(* PLC project mtcs_services, Institute of Astronomy OntoManager 0.0.1 *)
(* stored: creationDateTime 2017-02-05T17:05:48.277559, modificationDateTime 2017-02-05T17:05:48.277559 *)

TYPE ServicesTimingTimeSource : (LOCAL_CLOCK := 0, PTP_IEEE_1588 := 1);
END_TYPE

TYPE ServicesMeteoId : (WIND_SPEED_MINIMUM := 0, WIND_SPEED_AVERAGE := 1, WIND_SPEED_MAXIMUM := 2, WIND_DIRECTION_MINIMUM := 3, WIND_DIRECTION_AVERAGE := 4, WIND_DIRECTION_MAXIMUM := 5, AIR_PRESSURE := 6, AIR_TEMPERATURE := 7, INTERNAL_TEMPERATURE := 8, RELATIVE_HUMIDITY := 9, RAIN_ACCUMULATION := 10, RAIN_DURATION := 11, RAIN_INTENSITY := 12, RAIN_PEAK_INTENSITY := 13, HAIL_ACCUMULATION := 14, HAIL_DURATION := 15, HAIL_PEAK_INTENSITY := 16, HAIL_INTENSITY := 17, HEATING_TEMPERATURE := 18, HEATING_VOLTAGE := 19, SUPPLY_VOLTAGE := 20, REFERENCE_VOLTAGE := 21);
END_TYPE

TYPE ServicesParts : STRUCT
  timing : ServicesTiming;  (* Timing service *)
  meteo : ServicesMeteo;  (* Meteo service *)
  io : ServicesIO;  (* I/O modules *)
  configManager : ConfigManager;  (* The config manager (to load/save/activate configuration data) *)
END_STRUCT;
END_TYPE

TYPE ServicesTimingParts : STRUCT
  serialInfo : ServicesTimingSerialInfo;  (* Info acquired by serial link *)
END_STRUCT;
END_TYPE

TYPE ServicesIOParts : STRUCT
  coupler : EtherCatDevice;  (* Coupler *)
  slot1 : EtherCatDevice;  (* Slot 1 *)
  slot2 : EtherCatDevice;  (* Slot 2 *)
  slot3 : EtherCatDevice;  (* Slot 2 *)
END_STRUCT;
END_TYPE

TYPE ServicesProcesses : STRUCT
  initialize : Process;  (* Start initializing *)
  lock : Process;  (* Lock the system *)
  unlock : Process;  (* Unlock the system *)
  changeOperatingState : ChangeOperatingStateProcess;  (* Change the operating state (e.g. AUTO, MANUAL, ...) *)
END_STRUCT;
END_TYPE

TYPE ServicesTimingProcesses : STRUCT

END_STRUCT;
END_TYPE

TYPE ServicesMeteoProcesses : STRUCT

END_STRUCT;
END_TYPE

TYPE ServicesStatuses : STRUCT
  initializationStatus : InitializationStatus;
  healthStatus : HealthStatus;
  busyStatus : BusyStatus;
  operatingStatus : OperatingStatus;
END_STRUCT;
END_TYPE

TYPE ServicesTimingStatuses : STRUCT
  healthStatus : HealthStatus;
END_STRUCT;
END_TYPE

TYPE ServicesTimingSerialInfoStatuses : STRUCT
  portHealthStatus : HealthStatus;
  transmissionHealthStatus : HealthStatus;
  checksumHealthStatus : HealthStatus;
  healthStatus : HealthStatus;
END_STRUCT;
END_TYPE

TYPE ServicesMeteoMeasurementStatuses : STRUCT
  enabledStatus : EnabledStatus;  (* Is the temperature being measured? *)
  healthStatus : HealthStatus;  (* Is the data valid and within range? *)
  alarmStatus : HiHiLoLoAlarmStatus;  (* Alarm status *)
END_STRUCT;
END_TYPE

TYPE ServicesMeteoStatuses : STRUCT
  meteoHealthStatus : HealthStatus;
  healthStatus : HealthStatus;
END_STRUCT;
END_TYPE

TYPE ServicesIOStatuses : STRUCT
  healthStatus : HealthStatus;  (* Is the I/O in a healthy state? *)
END_STRUCT;
END_TYPE

TYPE ServicesTimingConfig : STRUCT
  leapSeconds : INT;  (* Number of leap seconds, so that UTC = TAI + this value. See ftp://maia.usno.navy.mil/ser7/tai-utc.dat for the latest number. *)
  dut : LREAL;  (* Delta UT (= UT1 - UTC). Put to 0.0 to ignore. *)
  alwaysUseLocalClock : BOOL;  (* If TRUE, then the local clock (source=LOCAL_CLOCK) will be used even if an external (more accurate!) clock is available *)
  ignoreSerialError : BOOL;  (* Don't show the Servicestiming status as ERROR in case the serial link fails *)
END_STRUCT;
END_TYPE

TYPE ServicesMeteoConfig : STRUCT
  wetLimit : LREAL;  (* Wet if (rainIntensity+hailIntrelaensity)>wetLimit *)
  windSpeedMinimum : MeasurementConfig;  (* Config for the wind speed minimum *)
  windSpeedAverage : MeasurementConfig;  (* Config for the wind speed average *)
  windSpeedMaximum : MeasurementConfig;  (* Config for the wind speed maximum *)
  windDirectionMinimum : MeasurementConfig;  (* Config for the wind direction minimum *)
  windDirectionAverage : MeasurementConfig;  (* Config for the wind direction average *)
  windDirectionMaximum : MeasurementConfig;  (* Config for the wind direction maximum *)
  airPressure : MeasurementConfig;  (* Config for the air pressure *)
  airTemperature : MeasurementConfig;  (* Config for the air temperature *)
  internalTemperature : MeasurementConfig;  (* Config for the internal temperature *)
  relativeHumidity : MeasurementConfig;  (* Config for the relative humidity *)
  rainAccumulation : MeasurementConfig;  (* Config for the rain accumulation *)
  rainDuration : MeasurementConfig;  (* Config for the rain duration *)
  rainIntensity : MeasurementConfig;  (* Config for the rain intensity *)
  rainPeakIntensity : MeasurementConfig;  (* Config for the rain peak intensity *)
  hailAccumulation : MeasurementConfig;  (* Config for the hail accumulation *)
  hailDuration : MeasurementConfig;  (* Config for the hail duration *)
  hailIntensity : MeasurementConfig;  (* Config for the hail intensity *)
  hailPeakIntensity : MeasurementConfig;  (* Config for the hail peak intensity *)
  heatingTemperature : MeasurementConfig;  (* Config for the heating temperature *)
  heatingVoltage : MeasurementConfig;  (* Config for the heating voltage *)
  supplyVoltage : MeasurementConfig;  (* Config for the supply voltage *)
  referenceVoltage : MeasurementConfig;  (* Config for the 3.5 V reference voltage *)
END_STRUCT;
END_TYPE

TYPE ServicesConfig : STRUCT
  timing : ServicesTimingConfig;  (* Timing config *)
  meteo : ServicesMeteoConfig;  (* Meteo config *)
END_STRUCT;
END_TYPE

FUNCTION_BLOCK SM_Services
  VAR_INPUT
    {attribute 'OPC.UA.DA' := '1'}
    {attribute 'OPC.UA.DA.Access' := '1'}
    editableConfig : ServicesConfig;  (* Editable configuration of the Services subsystem *)
  END_VAR
  VAR_OUTPUT
    {attribute 'OPC.UA.DA' := '1'}
    {attribute 'OPC.UA.DA.Access' := '1'}
    actualStatus : STRING;  (* Current status description *)
    previousStatus : STRING;  (* Previous status description *)
    {attribute 'OPC.UA.DA' := '1'}
    {attribute 'OPC.UA.DA.Access' := '1'}
    config : ServicesConfig;  (* Active configuration of the Services subsystem *)
    statuses : ServicesStatuses;  (* Statuses of the state machine *)
    parts : ServicesParts;  (* Parts of the state machine *)
    processes : ServicesProcesses;  (* Processes of the state machine *)
  END_VAR
  VAR_IN_OUT
    {attribute 'OPC.UA.DA' := '0'}
    operatorStatus : OperatorStatus;  (* Shared operator status *)
  END_VAR

            parts.timing(
    operatorStatus := operatorStatus,
    config := config.timing);
parts.meteo( config := config.meteo );
parts.io();
parts.configManager( isEnabled := operatorStatus.tech );
statuses.initializationStatus();
statuses.healthStatus(
    isGood := parts.timing.statuses.healthStatus.isGood AND (parts.meteo.statuses.healthStatus.isGood AND parts.io.statuses.healthStatus.isGood),
    hasWarning := parts.timing.statuses.healthStatus.hasWarning OR (parts.meteo.statuses.healthStatus.hasWarning OR parts.io.statuses.healthStatus.hasWarning));
statuses.busyStatus( isBusy := statuses.initializationStatus.initializing );
statuses.operatingStatus( superState := statuses.initializationStatus.initialized );
processes.initialize( isEnabled := statuses.initializationStatus.shutdown OR (statuses.initializationStatus.initializingFailed OR statuses.initializationStatus.initialized) );
processes.lock( isEnabled := operatorStatus.tech AND statuses.initializationStatus.initialized );
processes.unlock( isEnabled := operatorStatus.tech AND statuses.initializationStatus.locked );
processes.changeOperatingState( isEnabled := FALSE );

          

{attribute 'TcRpcEnable' := '1'}
METHOD initialize : RequestResults
                  initialize := THIS^.processes.initialize.request();

                
END_METHOD

{attribute 'TcRpcEnable' := '1'}
METHOD lock : RequestResults
                  lock := THIS^.processes.lock.request();

                
END_METHOD

{attribute 'TcRpcEnable' := '1'}
METHOD unlock : RequestResults
                  unlock := THIS^.processes.unlock.request();

                
END_METHOD

{attribute 'TcRpcEnable' := '1'}
METHOD changeOperatingState : RequestResults
  VAR_INPUT
    state : OperatingStates;
  END_VAR
                  changeOperatingState := THIS^.processes.changeOperatingState.request( state := state );

                
END_METHOD

{attribute 'TcRpcEnable' := '1'}
METHOD _log : BOOL
  VAR_INPUT
    name : STRING;  (* Name of this function block instance *)
  END_VAR
  VAR_IN_OUT
    buffer : LogBuffer;  (* Buffer to write all logging to *)
  END_VAR
  VAR
    subBuffer : LogBuffer;  (* Temporary buffer to write logging by parts (sub-statemachines) to *)
  END_VAR
                  THIS^.parts.timing._log(
    name := 'timing',
    buffer := subBuffer);
THIS^.parts.meteo._log(
    name := 'meteo',
    buffer := subBuffer);
THIS^.parts.io._log(
    name := 'io',
    buffer := subBuffer);
THIS^.parts.configManager._log(
    name := 'configManager',
    buffer := subBuffer);
LOGGER(
    name := name,
    actualStatus := THIS^.actualStatus,
    previousStatus := THIS^.previousStatus,
    buffer := buffer,
    subBuffer := subBuffer,
    pHealthStatus := ADR(THIS^.statuses.healthStatus),
    pBusyStatus := ADR(THIS^.statuses.busyStatus));

                
END_METHOD
END_FUNCTION_BLOCK

FUNCTION_BLOCK SM_ServicesTiming
  VAR_INPUT
    {attribute 'OPC.UA.DA' := '1'}
    {attribute 'OPC.UA.DA.Access' := '1'}
    fromEL6688 AT %I* : TmcFromIoEL6688;  (* Data from the EL6688 *)
    {attribute 'OPC.UA.DA' := '1'}
    {attribute 'OPC.UA.DA.Access' := '1'}
    fromEcatMaster AT %I* : TmcFromIoEcatMaster;  (* Data from the EtherCAT master *)
    {attribute 'OPC.UA.DA' := '1'}
    {attribute 'OPC.UA.DA.Access' := '1'}
    fromCppTiming AT %I* : TmcToPlcTiming;  (* Data from the C++ task *)
  END_VAR
  VAR_OUTPUT
    {attribute 'OPC.UA.DA' := '1'}
    {attribute 'OPC.UA.DA.Access' := '1'}
    actualStatus : STRING;  (* Current status description *)
    previousStatus : STRING;  (* Previous status description *)
    {attribute 'OPC.UA.DA' := '1'}
    {attribute 'OPC.UA.DA.Access' := '1'}
    toCppTiming AT %Q* : TmcFromPlcTiming;  (* Data to the C++ task *)
    {attribute 'OPC.UA.DA' := '1'}
    {attribute 'OPC.UA.DA.Access' := '1'}
    utcDateString : STRING;  (* UTC date as a string of format YYYY-MM-DD *)
    {attribute 'OPC.UA.DA' := '1'}
    {attribute 'OPC.UA.DA.Access' := '1'}
    utcTimeString : STRING;  (* UTC time as a string of format HH-MM-SS.SSS *)
    {attribute 'OPC.UA.DA' := '1'}
    {attribute 'OPC.UA.DA.Access' := '1'}
    internalTimestampString : STRING;  (* String representation of the internal timestamp *)
    {attribute 'OPC.UA.DA' := '1'}
    {attribute 'OPC.UA.DA.Access' := '1'}
    externalTimestampString : STRING;  (* String representation of the external timestamp (note: this is TAI, not UTC!) *)
    statuses : ServicesTimingStatuses;  (* Statuses of the state machine *)
    parts : ServicesTimingParts;  (* Parts of the state machine *)
    processes : ServicesTimingProcesses;  (* Processes of the state machine *)
  END_VAR
  VAR_IN_OUT
    {attribute 'OPC.UA.DA' := '0'}
    operatorStatus : OperatorStatus;  (* Shared operator status *)
    {attribute 'OPC.UA.DA' := '0'}
    config : ServicesTimingConfig;  (* The config *)
  END_VAR

            parts.serialInfo();
statuses.healthStatus( isGood := config.ignoreSerialError OR parts.serialInfo.statuses.healthStatus.good );

          

{attribute 'TcRpcEnable' := '1'}
METHOD _log : BOOL
  VAR_INPUT
    name : STRING;  (* Name of this function block instance *)
  END_VAR
  VAR_IN_OUT
    buffer : LogBuffer;  (* Buffer to write all logging to *)
  END_VAR
  VAR
    subBuffer : LogBuffer;  (* Temporary buffer to write logging by parts (sub-statemachines) to *)
  END_VAR
                  THIS^.parts.serialInfo._log(
    name := 'serialInfo',
    buffer := subBuffer);
LOGGER(
    name := name,
    actualStatus := THIS^.actualStatus,
    previousStatus := THIS^.previousStatus,
    buffer := buffer,
    subBuffer := subBuffer,
    pHealthStatus := ADR(THIS^.statuses.healthStatus));

                
END_METHOD
END_FUNCTION_BLOCK

FUNCTION_BLOCK SM_ServicesTimingSerialInfo
  VAR_OUTPUT
    {attribute 'OPC.UA.DA' := '1'}
    {attribute 'OPC.UA.DA.Access' := '1'}
    actualStatus : STRING;  (* Current status description *)
    previousStatus : STRING;  (* Previous status description *)
    {attribute 'OPC.UA.DA' := '1'}
    {attribute 'OPC.UA.DA.Access' := '1'}
    serialTimeout : BOOL;  (* Is the serial data not being received within time? *)
    {attribute 'OPC.UA.DA' := '1'}
    {attribute 'OPC.UA.DA.Access' := '1'}
    comError : BOOL;  (* Is there any problem with the COM port? *)
    {attribute 'OPC.UA.DA' := '1'}
    {attribute 'OPC.UA.DA.Access' := '1'}
    comErrorID : INT;  (* COM error id (see Beckhoff ComError_t) *)
    {attribute 'OPC.UA.DA' := '1'}
    {attribute 'OPC.UA.DA.Access' := '1'}
    comErrorDescription : STRING;  (* Description of the COM error id *)
    {attribute 'OPC.UA.DA' := '1'}
    {attribute 'OPC.UA.DA.Access' := '1'}
    time_h : USINT;  (* Time: hours (0-24) *)
    {attribute 'OPC.UA.DA' := '1'}
    {attribute 'OPC.UA.DA.Access' := '1'}
    time_m : USINT;  (* Time: minutes (0-59) *)
    {attribute 'OPC.UA.DA' := '1'}
    {attribute 'OPC.UA.DA.Access' := '1'}
    time_s : USINT;  (* Time: seconds (0-59, or 60 if leap second) *)
    {attribute 'OPC.UA.DA' := '1'}
    {attribute 'OPC.UA.DA.Access' := '1'}
    latitude_deg : USINT;  (* Latitude: degrees (0-90) *)
    {attribute 'OPC.UA.DA' := '1'}
    {attribute 'OPC.UA.DA.Access' := '1'}
    latitude_min : REAL;  (* Latitude: minutes (0.0-59.99999) *)
    {attribute 'OPC.UA.DA' := '1'}
    {attribute 'OPC.UA.DA.Access' := '1'}
    latitude_sign : STRING;  (* Latitude: sign (either 'N' or 'S') *)
    {attribute 'OPC.UA.DA' := '1'}
    {attribute 'OPC.UA.DA.Access' := '1'}
    longitude_deg : USINT;  (* Longitude: degrees (0-180) *)
    {attribute 'OPC.UA.DA' := '1'}
    {attribute 'OPC.UA.DA.Access' := '1'}
    longitude_min : REAL;  (* Longitude: minutes (0.0-59.99999) *)
    {attribute 'OPC.UA.DA' := '1'}
    {attribute 'OPC.UA.DA.Access' := '1'}
    longitude_sign : STRING;  (* Longitude: sign (either 'E' or 'W') *)
    {attribute 'OPC.UA.DA' := '1'}
    {attribute 'OPC.UA.DA.Access' := '1'}
    positionFix : BOOL;  (* True if a position fix was accomplished, False if not *)
    {attribute 'OPC.UA.DA' := '1'}
    {attribute 'OPC.UA.DA.Access' := '1'}
    satellitesUsed : USINT;  (* Number of satellites used *)
    {attribute 'OPC.UA.DA' := '1'}
    {attribute 'OPC.UA.DA.Access' := '1'}
    horizontalDilutionOfPosition : REAL;  (* Horizontal dilution of position *)
    {attribute 'OPC.UA.DA' := '1'}
    {attribute 'OPC.UA.DA.Access' := '1'}
    meanSeaLevelAltitude : REAL;  (* Mean altitude above sea level in meters *)
    {attribute 'OPC.UA.DA' := '1'}
    {attribute 'OPC.UA.DA.Access' := '1'}
    geoidSeparation : REAL;  (* Geoid separation in meters *)
    {attribute 'OPC.UA.DA' := '1'}
    {attribute 'OPC.UA.DA.Access' := '1'}
    checksum : USINT;  (* Checksum send by the time server *)
    {attribute 'OPC.UA.DA' := '1'}
    {attribute 'OPC.UA.DA.Access' := '1'}
    calculatedChecksum : USINT;  (* Checksum calculated by the PLC *)
    statuses : ServicesTimingSerialInfoStatuses;  (* Statuses of the state machine *)
  END_VAR

            statuses.portHealthStatus( isGood := NOT(comError) );
statuses.transmissionHealthStatus( isGood := NOT(serialTimeout) );
statuses.checksumHealthStatus( isGood := checksum = calculatedChecksum );
statuses.healthStatus( isGood := statuses.portHealthStatus.good AND (statuses.transmissionHealthStatus.good AND statuses.checksumHealthStatus.good) );

          

{attribute 'TcRpcEnable' := '1'}
METHOD _log : BOOL
  VAR_INPUT
    name : STRING;  (* Name of this function block instance *)
  END_VAR
  VAR_IN_OUT
    buffer : LogBuffer;  (* Buffer to write all logging to *)
  END_VAR
  VAR
    subBuffer : LogBuffer;  (* Temporary buffer to write logging by parts (sub-statemachines) to *)
  END_VAR
                  LOGGER(
    name := name,
    actualStatus := THIS^.actualStatus,
    previousStatus := THIS^.previousStatus,
    buffer := buffer,
    subBuffer := subBuffer,
    pHealthStatus := ADR(THIS^.statuses.healthStatus));

                
END_METHOD
END_FUNCTION_BLOCK

FUNCTION_BLOCK SM_ServicesMeteoMeasurement
  VAR_INPUT
    {attribute 'OPC.UA.DA' := '1'}
    {attribute 'OPC.UA.DA.Access' := '1'}
    id : ServicesMeteoId;  (* ID *)
    {attribute 'OPC.UA.DA' := '0'}
    inputString : STRING;  (* Input string from the meteo station *)
  END_VAR
  VAR_OUTPUT
    {attribute 'OPC.UA.DA' := '1'}
    {attribute 'OPC.UA.DA.Access' := '1'}
    actualStatus : STRING;  (* Current status description *)
    previousStatus : STRING;  (* Previous status description *)
    {attribute 'OPC.UA.DA' := '1'}
    {attribute 'OPC.UA.DA.Access' := '1'}
    data : QuantityValue;  (* Actual value *)
    {attribute 'OPC.UA.DA' := '1'}
    {attribute 'OPC.UA.DA.Access' := '1'}
    invalidData : BOOL;  (* True if the data is invalid *)
    {attribute 'OPC.UA.DA' := '1'}
    {attribute 'OPC.UA.DA.Access' := '1'}
    lastChar : STRING;  (* Last character *)
    {attribute 'OPC.UA.DA' := '1'}
    {attribute 'OPC.UA.DA.Access' := '1'}
    name : STRING;  (* Name of the measurementw *)
    statuses : ServicesMeteoMeasurementStatuses;  (* Statuses of the state machine *)
  END_VAR
  VAR_IN_OUT
    {attribute 'OPC.UA.DA' := '0'}
    config : MeasurementConfig;  (* Reference to the config *)
  END_VAR

            statuses.enabledStatus( isEnabled := config.enabled );
statuses.healthStatus(
    superState := statuses.enabledStatus.enabled,
    isGood := NOT(invalidData OR (statuses.alarmStatus.hiHi OR statuses.alarmStatus.loLo)),
    hasWarning := statuses.alarmStatus.hi OR statuses.alarmStatus.lo);
statuses.alarmStatus(
    superState := statuses.enabledStatus.enabled,
    config := config.alarms,
    value := data.value);

          

{attribute 'TcRpcEnable' := '1'}
METHOD _log : BOOL
  VAR_INPUT
    name : STRING;  (* Name of this function block instance *)
  END_VAR
  VAR_IN_OUT
    buffer : LogBuffer;  (* Buffer to write all logging to *)
  END_VAR
  VAR
    subBuffer : LogBuffer;  (* Temporary buffer to write logging by parts (sub-statemachines) to *)
  END_VAR
                  LOGGER(
    name := name,
    actualStatus := THIS^.actualStatus,
    previousStatus := THIS^.previousStatus,
    buffer := buffer,
    subBuffer := subBuffer,
    pHealthStatus := ADR(THIS^.statuses.healthStatus));

                
END_METHOD
END_FUNCTION_BLOCK

FUNCTION_BLOCK SM_ServicesMeteo
  VAR_INPUT
    {attribute 'OPC.UA.DA' := '1'}
    {attribute 'OPC.UA.DA.Access' := '1'}
    serialTimeout : BOOL;  (* Is the serial data not being received within time? *)
    {attribute 'OPC.UA.DA' := '1'}
    {attribute 'OPC.UA.DA.Access' := '1'}
    comError : BOOL;  (* Is there any problem with the COM port? *)
    {attribute 'OPC.UA.DA' := '1'}
    {attribute 'OPC.UA.DA.Access' := '1'}
    comErrorID : INT;  (* COM error id (see Beckhoff ComError_t) *)
    {attribute 'OPC.UA.DA' := '1'}
    {attribute 'OPC.UA.DA.Access' := '1'}
    comErrorDescription : STRING;  (* Description of the COM error id *)
    {attribute 'OPC.UA.DA' := '1'}
    {attribute 'OPC.UA.DA.Access' := '1'}
    windSpeedMinimum : ServicesMeteoMeasurement;  (* Wind speed minimum *)
    {attribute 'OPC.UA.DA' := '1'}
    {attribute 'OPC.UA.DA.Access' := '1'}
    windSpeedAverage : ServicesMeteoMeasurement;  (* Wind speed average *)
    {attribute 'OPC.UA.DA' := '1'}
    {attribute 'OPC.UA.DA.Access' := '1'}
    windSpeedMaximum : ServicesMeteoMeasurement;  (* Wind speed maximum *)
    {attribute 'OPC.UA.DA' := '1'}
    {attribute 'OPC.UA.DA.Access' := '1'}
    windDirectionMinimum : ServicesMeteoMeasurement;  (* Wind direction minimum *)
    {attribute 'OPC.UA.DA' := '1'}
    {attribute 'OPC.UA.DA.Access' := '1'}
    windDirectionAverage : ServicesMeteoMeasurement;  (* Wind direction average *)
    {attribute 'OPC.UA.DA' := '1'}
    {attribute 'OPC.UA.DA.Access' := '1'}
    windDirectionMaximum : ServicesMeteoMeasurement;  (* Wind direction maximum *)
    {attribute 'OPC.UA.DA' := '1'}
    {attribute 'OPC.UA.DA.Access' := '1'}
    airPressure : ServicesMeteoMeasurement;  (* Air pressure *)
    {attribute 'OPC.UA.DA' := '1'}
    {attribute 'OPC.UA.DA.Access' := '1'}
    airTemperature : ServicesMeteoMeasurement;  (* Air temperature *)
    {attribute 'OPC.UA.DA' := '1'}
    {attribute 'OPC.UA.DA.Access' := '1'}
    internalTemperature : ServicesMeteoMeasurement;  (* Internal temperature *)
    {attribute 'OPC.UA.DA' := '1'}
    {attribute 'OPC.UA.DA.Access' := '1'}
    relativeHumidity : ServicesMeteoMeasurement;  (* Relative humidity *)
    {attribute 'OPC.UA.DA' := '1'}
    {attribute 'OPC.UA.DA.Access' := '1'}
    rainAccumulation : ServicesMeteoMeasurement;  (* Rain accumulation *)
    {attribute 'OPC.UA.DA' := '1'}
    {attribute 'OPC.UA.DA.Access' := '1'}
    rainDuration : ServicesMeteoMeasurement;  (* Rain duration *)
    {attribute 'OPC.UA.DA' := '1'}
    {attribute 'OPC.UA.DA.Access' := '1'}
    rainIntensity : ServicesMeteoMeasurement;  (* Rain intensity *)
    {attribute 'OPC.UA.DA' := '1'}
    {attribute 'OPC.UA.DA.Access' := '1'}
    rainPeakIntensity : ServicesMeteoMeasurement;  (* Rain peak intensity *)
    {attribute 'OPC.UA.DA' := '1'}
    {attribute 'OPC.UA.DA.Access' := '1'}
    hailAccumulation : ServicesMeteoMeasurement;  (* Hail accumulation *)
    {attribute 'OPC.UA.DA' := '1'}
    {attribute 'OPC.UA.DA.Access' := '1'}
    hailDuration : ServicesMeteoMeasurement;  (* Hail duration *)
    {attribute 'OPC.UA.DA' := '1'}
    {attribute 'OPC.UA.DA.Access' := '1'}
    hailIntensity : ServicesMeteoMeasurement;  (* Hail intensity *)
    {attribute 'OPC.UA.DA' := '1'}
    {attribute 'OPC.UA.DA.Access' := '1'}
    hailPeakIntensity : ServicesMeteoMeasurement;  (* Hail peak intensity *)
    {attribute 'OPC.UA.DA' := '1'}
    {attribute 'OPC.UA.DA.Access' := '1'}
    heatingTemperature : ServicesMeteoMeasurement;  (* Heating temperature *)
    {attribute 'OPC.UA.DA' := '1'}
    {attribute 'OPC.UA.DA.Access' := '1'}
    heatingVoltage : ServicesMeteoMeasurement;  (* Heating voltage *)
    {attribute 'OPC.UA.DA' := '1'}
    {attribute 'OPC.UA.DA.Access' := '1'}
    supplyVoltage : ServicesMeteoMeasurement;  (* Supply voltage *)
    {attribute 'OPC.UA.DA' := '1'}
    {attribute 'OPC.UA.DA.Access' := '1'}
    referenceVoltage : ServicesMeteoMeasurement;  (* Reference voltage *)
    {attribute 'OPC.UA.DA' := '1'}
    {attribute 'OPC.UA.DA.Access' := '1'}
    durationOK : Duration;  (* Duration that the meteo is OK *)
    {attribute 'OPC.UA.DA' := '1'}
    {attribute 'OPC.UA.DA.Access' := '1'}
    dewpoint : Temperature;  (* Calculated dewpoint *)
    {attribute 'OPC.UA.DA' := '1'}
    {attribute 'OPC.UA.DA.Access' := '1'}
    wet : BOOL;  (* Wet if (rainIntensity+hailIntensity) > config.wetLimit *)
    {attribute 'OPC.UA.DA' := '1'}
    {attribute 'OPC.UA.DA.Access' := '1'}
    heating : BOOL;  (* Heating or not? *)
    {attribute 'OPC.UA.DA' := '1'}
    {attribute 'OPC.UA.DA.Access' := '1'}
    windDirectionMinimumString : STRING;  (* Average direction of the wind as a string *)
    {attribute 'OPC.UA.DA' := '1'}
    {attribute 'OPC.UA.DA.Access' := '1'}
    windDirectionAverageString : STRING;  (* Average direction of the wind as a string *)
    {attribute 'OPC.UA.DA' := '1'}
    {attribute 'OPC.UA.DA.Access' := '1'}
    windDirectionMaximumString : STRING;  (* Average direction of the wind as a string *)
  END_VAR
  VAR_OUTPUT
    {attribute 'OPC.UA.DA' := '1'}
    {attribute 'OPC.UA.DA.Access' := '1'}
    actualStatus : STRING;  (* Current status description *)
    previousStatus : STRING;  (* Previous status description *)
    statuses : ServicesMeteoStatuses;  (* Statuses of the state machine *)
    processes : ServicesMeteoProcesses;  (* Processes of the state machine *)
  END_VAR
  VAR_IN_OUT
    {attribute 'OPC.UA.DA' := '0'}
    config : ServicesMeteoConfig;  (* The config *)
  END_VAR

            windSpeedMinimum(
    id := ServicesMeteoId.WIND_SPEED_MINIMUM,
    config := config.windSpeedMinimum);
windSpeedAverage(
    id := ServicesMeteoId.WIND_SPEED_AVERAGE,
    config := config.windSpeedAverage);
windSpeedMaximum(
    id := ServicesMeteoId.WIND_SPEED_MAXIMUM,
    config := config.windSpeedMaximum);
windDirectionMinimum(
    id := ServicesMeteoId.WIND_DIRECTION_MINIMUM,
    config := config.windDirectionMinimum);
windDirectionAverage(
    id := ServicesMeteoId.WIND_DIRECTION_AVERAGE,
    config := config.windDirectionAverage);
windDirectionMaximum(
    id := ServicesMeteoId.WIND_DIRECTION_MAXIMUM,
    config := config.windDirectionMaximum);
airPressure(
    id := ServicesMeteoId.AIR_PRESSURE,
    config := config.airPressure);
airTemperature(
    id := ServicesMeteoId.AIR_TEMPERATURE,
    config := config.airTemperature);
internalTemperature(
    id := ServicesMeteoId.INTERNAL_TEMPERATURE,
    config := config.internalTemperature);
relativeHumidity(
    id := ServicesMeteoId.RELATIVE_HUMIDITY,
    config := config.relativeHumidity);
rainAccumulation(
    id := ServicesMeteoId.RAIN_ACCUMULATION,
    config := config.rainAccumulation);
rainDuration(
    id := ServicesMeteoId.RAIN_DURATION,
    config := config.rainDuration);
rainIntensity(
    id := ServicesMeteoId.RAIN_INTENSITY,
    config := config.rainIntensity);
rainPeakIntensity(
    id := ServicesMeteoId.RAIN_PEAK_INTENSITY,
    config := config.rainPeakIntensity);
hailAccumulation(
    id := ServicesMeteoId.HAIL_ACCUMULATION,
    config := config.hailAccumulation);
hailDuration(
    id := ServicesMeteoId.HAIL_DURATION,
    config := config.hailDuration);
hailIntensity(
    id := ServicesMeteoId.HAIL_INTENSITY,
    config := config.hailIntensity);
hailPeakIntensity(
    id := ServicesMeteoId.HAIL_PEAK_INTENSITY,
    config := config.hailPeakIntensity);
heatingTemperature(
    id := ServicesMeteoId.HEATING_TEMPERATURE,
    config := config.heatingTemperature);
heatingVoltage(
    id := ServicesMeteoId.HEATING_VOLTAGE,
    config := config.heatingVoltage);
supplyVoltage(
    id := ServicesMeteoId.SUPPLY_VOLTAGE,
    config := config.supplyVoltage);
referenceVoltage(
    id := ServicesMeteoId.REFERENCE_VOLTAGE,
    config := config.referenceVoltage);
statuses.meteoHealthStatus(
    superState := statuses.healthStatus.good,
    isGood := (windSpeedMinimum.statuses.healthStatus.isGood OR windSpeedMinimum.statuses.enabledStatus.disabled) AND ((windSpeedAverage.statuses.healthStatus.isGood OR windSpeedAverage.statuses.enabledStatus.disabled) AND ((windSpeedMaximum.statuses.healthStatus.isGood OR windSpeedMaximum.statuses.enabledStatus.disabled) AND ((windDirectionMinimum.statuses.healthStatus.isGood OR windDirectionMinimum.statuses.enabledStatus.disabled) AND ((windDirectionAverage.statuses.healthStatus.isGood OR windDirectionAverage.statuses.enabledStatus.disabled) AND ((windDirectionMaximum.statuses.healthStatus.isGood OR windDirectionMaximum.statuses.enabledStatus.disabled) AND ((airPressure.statuses.healthStatus.isGood OR airPressure.statuses.enabledStatus.disabled) AND ((airTemperature.statuses.healthStatus.isGood OR airTemperature.statuses.enabledStatus.disabled) AND ((internalTemperature.statuses.healthStatus.isGood OR internalTemperature.statuses.enabledStatus.disabled) AND ((relativeHumidity.statuses.healthStatus.isGood OR relativeHumidity.statuses.enabledStatus.disabled) AND ((rainAccumulation.statuses.healthStatus.isGood OR rainAccumulation.statuses.enabledStatus.disabled) AND ((rainDuration.statuses.healthStatus.isGood OR rainDuration.statuses.enabledStatus.disabled) AND ((rainIntensity.statuses.healthStatus.isGood OR rainIntensity.statuses.enabledStatus.disabled) AND ((rainPeakIntensity.statuses.healthStatus.isGood OR rainPeakIntensity.statuses.enabledStatus.disabled) AND ((hailAccumulation.statuses.healthStatus.isGood OR hailAccumulation.statuses.enabledStatus.disabled) AND ((hailDuration.statuses.healthStatus.isGood OR hailDuration.statuses.enabledStatus.disabled) AND ((hailIntensity.statuses.healthStatus.isGood OR hailIntensity.statuses.enabledStatus.disabled) AND ((hailPeakIntensity.statuses.healthStatus.isGood OR hailPeakIntensity.statuses.enabledStatus.disabled) AND ((heatingTemperature.statuses.healthStatus.isGood OR heatingTemperature.statuses.enabledStatus.disabled) AND ((heatingVoltage.statuses.healthStatus.isGood OR heatingVoltage.statuses.enabledStatus.disabled) AND ((supplyVoltage.statuses.healthStatus.isGood OR supplyVoltage.statuses.enabledStatus.disabled) AND (referenceVoltage.statuses.healthStatus.isGood OR referenceVoltage.statuses.enabledStatus.disabled))))))))))))))))))))),
    hasWarning := windSpeedMinimum.statuses.healthStatus.hasWarning OR (windSpeedAverage.statuses.healthStatus.hasWarning OR (windSpeedMaximum.statuses.healthStatus.hasWarning OR (windDirectionMinimum.statuses.healthStatus.hasWarning OR (windDirectionAverage.statuses.healthStatus.hasWarning OR (windDirectionMaximum.statuses.healthStatus.hasWarning OR (airPressure.statuses.healthStatus.hasWarning OR (airTemperature.statuses.healthStatus.hasWarning OR (internalTemperature.statuses.healthStatus.hasWarning OR (relativeHumidity.statuses.healthStatus.hasWarning OR (rainAccumulation.statuses.healthStatus.hasWarning OR (rainDuration.statuses.healthStatus.hasWarning OR (rainIntensity.statuses.healthStatus.hasWarning OR (rainPeakIntensity.statuses.healthStatus.hasWarning OR (hailAccumulation.statuses.healthStatus.hasWarning OR (hailDuration.statuses.healthStatus.hasWarning OR (hailIntensity.statuses.healthStatus.hasWarning OR (hailPeakIntensity.statuses.healthStatus.hasWarning OR (heatingTemperature.statuses.healthStatus.hasWarning OR (heatingVoltage.statuses.healthStatus.hasWarning OR (supplyVoltage.statuses.healthStatus.hasWarning OR referenceVoltage.statuses.healthStatus.hasWarning)))))))))))))))))))));
statuses.healthStatus( isGood := NOT(serialTimeout OR comError) );

          

{attribute 'TcRpcEnable' := '1'}
METHOD _log : BOOL
  VAR_INPUT
    name : STRING;  (* Name of this function block instance *)
  END_VAR
  VAR_IN_OUT
    buffer : LogBuffer;  (* Buffer to write all logging to *)
  END_VAR
  VAR
    subBuffer : LogBuffer;  (* Temporary buffer to write logging by parts (sub-statemachines) to *)
  END_VAR
                  LOGGER(
    name := name,
    actualStatus := THIS^.actualStatus,
    previousStatus := THIS^.previousStatus,
    buffer := buffer,
    subBuffer := subBuffer,
    pHealthStatus := ADR(THIS^.statuses.healthStatus));

                
END_METHOD
END_FUNCTION_BLOCK

FUNCTION_BLOCK SM_ServicesIO
  VAR_OUTPUT
    {attribute 'OPC.UA.DA' := '1'}
    {attribute 'OPC.UA.DA.Access' := '1'}
    actualStatus : STRING;  (* Current status description *)
    previousStatus : STRING;  (* Previous status description *)
    statuses : ServicesIOStatuses;  (* Statuses of the state machine *)
    parts : ServicesIOParts;  (* Parts of the state machine *)
  END_VAR

            parts.coupler(
    id := 'COUPLER',
    typeId := 'EK1100');
parts.slot1(
    id := 'TI-RS232',
    typeId := 'EL6001');
parts.slot2(
    id := 'METEO',
    typeId := 'EL6001');
parts.slot3(
    id := 'WESTS',
    typeId := 'EL6001');
statuses.healthStatus( isGood := parts.coupler.statuses.healthStatus.isGood AND (parts.slot1.statuses.healthStatus.isGood AND parts.slot2.statuses.healthStatus.isGood) );

          

{attribute 'TcRpcEnable' := '1'}
METHOD _log : BOOL
  VAR_INPUT
    name : STRING;  (* Name of this function block instance *)
  END_VAR
  VAR_IN_OUT
    buffer : LogBuffer;  (* Buffer to write all logging to *)
  END_VAR
  VAR
    subBuffer : LogBuffer;  (* Temporary buffer to write logging by parts (sub-statemachines) to *)
  END_VAR
                  THIS^.parts.coupler._log(
    name := 'coupler',
    buffer := subBuffer);
THIS^.parts.slot1._log(
    name := 'slot1',
    buffer := subBuffer);
THIS^.parts.slot2._log(
    name := 'slot2',
    buffer := subBuffer);
THIS^.parts.slot3._log(
    name := 'slot3',
    buffer := subBuffer);
LOGGER(
    name := name,
    actualStatus := THIS^.actualStatus,
    previousStatus := THIS^.previousStatus,
    buffer := buffer,
    subBuffer := subBuffer,
    pHealthStatus := ADR(THIS^.statuses.healthStatus));

                
END_METHOD
END_FUNCTION_BLOCK
